PROGRAM MAIN
VAR
END_VAR

END_PROGRAM

(* stored: Version 1.1.0.1, ProductVersion 3.1.4024.12
   POU MAIN: Id {2ab8832a-ed8a-4e83-984d-fd75a1e41693}, SpecialFunc None *)
